// TIA Portal V19 export
TYPE "LAF_typeDevDiagAlarm"
TITLE = PN device diag alarms / Alarme PN-D<evice Diagnose
// This data type contains the structure of possible alarms. / Struktur Alarme PN-Device Diagnose
// stored: Access Published
   STRUCT
      invalidValueMaxDevices { ExternalAccessible := 'False'; ExternalVisible := 'False'; ExternalWritable := 'False'} : Bool;   // Ungueltiger Wert / Anwenderk. "PNDevDiag": MAX_NO_OF_DEVICES [1..] / Invalid Value / Userconstant "PNDevDiag": MAX_NO_OF_DEVICES [1..]
      invalidValueMaxModules { ExternalAccessible := 'False'; ExternalVisible := 'False'; ExternalWritable := 'False'} : Bool;   // Ungueltiger Wert / Anwenderk. "PNDevDiag": MAX_NO_OF_MODULES [1..128] / Invalid Value / Userconstant "PNDevDiag": MAX_NO_OF_MODULES [1..128]
      invalidAddressLog2Geo { ExternalAccessible := 'False'; ExternalVisible := 'False'; ExternalWritable := 'False'} : Bool;   // Ungueltige Adresse "PNDevDiag": LOG2GEO_LOCAL_PNIO-SYSTEM / Invalid Address "PNDevDiag": LOG2GEO_LOCAL_PNIO-SYSTEM
      errorReadDeviceStates { ExternalAccessible := 'False'; ExternalVisible := 'False'; ExternalWritable := 'False'} : Bool;   // PROFINET Geraete-Status: Fehler beim lesen des Geraetestatus / PROFINET Device-States: Error Read Device-States
      deviceFaulty { ExternalAccessible := 'False'; ExternalVisible := 'False'; ExternalWritable := 'False'} : Bool;   // PROFINET-Geraet ist gestoert / PROFINET-Device faulty
      deviceProblem { ExternalAccessible := 'False'; ExternalVisible := 'False'; ExternalWritable := 'False'} : Bool;   // PROFINET-Geraet meldet Problem / PROFINET-Device with Problem
      deviceDeactivated { ExternalAccessible := 'False'; ExternalVisible := 'False'; ExternalWritable := 'False'} : Bool;   // PROFINET-Geraet deaktiviert / PROFINET-Device deactivated
      deviceNotPresent { ExternalAccessible := 'False'; ExternalVisible := 'False'; ExternalWritable := 'False'} : Bool;   // PROFINET-Geraet nicht vorhanden, jedoch konfiguriert / PROFINET-Device not present but configured
      deviceNetworkError { ExternalAccessible := 'False'; ExternalVisible := 'False'; ExternalWritable := 'False'} : Bool;   // PROFINET-Geraet meldet Netzwerkfehler (z.B. Topologie-Fehler) / PROFINET-Device with network error (e.g. Topology-error)
      deviceMaintRequired { ExternalAccessible := 'False'; ExternalVisible := 'False'; ExternalWritable := 'False'} : Bool;   // POFINET-Geraet meldet Wartungsbedarf / POFINET-Device with maintenance demanded
      deviceMaintDemanded { ExternalAccessible := 'False'; ExternalVisible := 'False'; ExternalWritable := 'False'} : Bool;   // POFINET-Geraet meldet Wartungsanforderung / POFINET-Device with maintenance required
      spare11 { ExternalAccessible := 'False'; ExternalVisible := 'False'; ExternalWritable := 'False'} : Bool;   // Reserve11 / spare11
      spare12 { ExternalAccessible := 'False'; ExternalVisible := 'False'; ExternalWritable := 'False'} : Bool;   // Reserve12 / spare12
      spare13 { ExternalAccessible := 'False'; ExternalVisible := 'False'; ExternalWritable := 'False'} : Bool;   // Reserve13 / spare13
      spare14 { ExternalAccessible := 'False'; ExternalVisible := 'False'; ExternalWritable := 'False'} : Bool;   // Reserve14 / spare14
      spare15 { ExternalAccessible := 'False'; ExternalVisible := 'False'; ExternalWritable := 'False'} : Bool;   // Reserve15 / spare15
   END_STRUCT;
END_TYPE
